(* CoDeSys 2.3.9.37 project: Cap12_1.pro *)
(* Libraries: Standard.LIB 4.10.05 12:14:46 *)

(* POU PLC_PRG, FBD *)
PROGRAM PLC_PRG
VAR
	Escal_Input: Escalado;
	EntLogica: REAL;
	SalIngenieria: REAL;
	ErrorEscalado: BOOL;
END_VAR
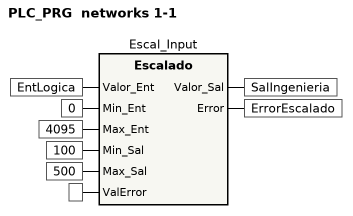
_FBD_ (* Function Block Diagram *)
NETWORK 1
	Escal_Input:Escalado(Valor_Ent: EntLogica, Min_Ent: 0, Max_Ent: 4095, Min_Sal: 100, Max_Sal: 500, ValError: , Error => ErrorEscalado) => SalIngenieria
_END_FBD_
END_PROGRAM

(* POU Escalado, ST *)
FUNCTION_BLOCK Escalado
VAR_INPUT
	Valor_Ent : REAL;    (* Valor a convertir *)
	Min_Ent : REAL;      (* Valor mínimo de la entrada *)
	Max_Ent : REAL;	  (* Valor máximo de la entrada *)
	Min_Sal : REAL;      (* Valor mínimo de la salida *)
	Max_Sal : REAL;	   (* . Valor máximo de la salida. *)
      ValError : REAL:=-1;    (*Valor al que poner la salida en caso de error. Por defecto -1*)
END_VAR
VAR_OUTPUT
	Valor_Sal : REAL;   (*. Valor convertido *)
	Error :  BOOL;         (* Se activa cuando el valor de entrada queda fuera de límites *)
END_VAR
VAR
	pendiente: REAL;
END_VAR
Error:= (Valor_Ent>Max_Ent) OR (Valor_Ent<Min_Ent);

IF NOT Error THEN
   pendiente:=(Max_Sal-Min_Sal)/(Max_Ent-Min_Ent);
   Valor_Sal:=Valor_Ent*pendiente+Min_Sal;
ELSE
   Valor_Sal:=ValError;
END_IF
END_FUNCTION_BLOCK

(* Visualisation Visu
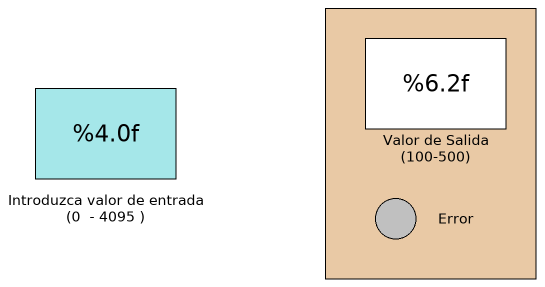
rectangle at (90,100)-(231,191): text "%4.0f"; shows PLC_PRG.EntLogica; editable
rectangle at (50,180)-(271,261): text "Introduzca valor de entrada / (0  - 4095 )"
rectangle at (420,50)-(561,141): text "%6.2f"; shows PLC_PRG.SalIngenieria
rectangle at (380,120)-(601,201): text "Valor de Salida / (100-500)"
ellipse at (430,210)-(471,251): alarm colour if PLC_PRG.ErrorEscalado
rectangle at (450,210)-(571,251): text "Error"
1 more shapes without text or variables
*)
